{attribute 'linkalways'} 
{attribute 'no_explicit_call' := 'This FB is a CLASS and must be accessed using methods or properties'}
{attribute 'enable_dynamic_creation'}
FUNCTION_BLOCK _ETcVnCircularityCalculationMethod EXTENDS EnumDatatypeBase
VAR
	localData : ETcVnCircularityCalculationMethod;
	activeData : REFERENCE TO ETcVnCircularityCalculationMethod;
	enumBaseDatatype : _DINT(localData);
END_VAR

METHOD PRIVATE AddLocalEnumeration
VAR_INPUT
	Enumeration : T_MAXSTRING;
	Value : ETcVnCircularityCalculationMethod;
END_VAR
AddEnumeration(Enumeration, Value);
END_METHOD

PROPERTY PUBLIC Address : PVOID
GET
Address := ADR(activeData);
END_GET
END_PROPERTY

METHOD PUBLIC ClearReference
VAR_INPUT
END_VAR
activeData REF= localData;
SetBaseDatatypeReference();
END_METHOD

METHOD PUBLIC Clone : I_Datatype
VAR
    pClone : POINTER TO _ETcVnCircularityCalculationMethod;
END_VAR
pClone := __NEW(_ETcVnCircularityCalculationMethod(InitialValue := Value));
Clone := pClone^;
END_METHOD

METHOD FB_init : BOOL
VAR_INPUT
	bInitRetains : BOOL; // if TRUE, the retain variables are initialized (warm start / cold start)
	bInCopyCode : BOOL;  // if TRUE, the instance afterwards gets moved into the copy code (online change)
	InitialValue : ETcVnCircularityCalculationMethod;
END_VAR
localData := InitialValue;
AddBaseDatatype(enumBaseDatatype);
ClearReference();

AddLocalEnumeration('TCVN_CCM_DEFAULT', ETcVnCircularityCalculationMethod.TCVN_CCM_DEFAULT);
AddLocalEnumeration('TCVN_CCM_CONVEXHULL_PERIMETER', ETcVnCircularityCalculationMethod.TCVN_CCM_CONVEXHULL_PERIMETER);
AddLocalEnumeration('TCVN_CCM_MAX_RADIUS', ETcVnCircularityCalculationMethod.TCVN_CCM_MAX_RADIUS);
AddLocalEnumeration('TCVN_CCM_ENCLOSINGCIRCLE_RADIUS', ETcVnCircularityCalculationMethod.TCVN_CCM_ENCLOSINGCIRCLE_RADIUS);
END_METHOD

PROPERTY PUBLIC Identifier : T_MAXSTRING
GET
Identifier := 'ETcVnCircularityCalculationMethod';
END_GET
END_PROPERTY

METHOD IsEnumeratorValueEqual : BOOL
VAR_INPUT
	Enumerator : I_KeyValueForwardEnumerator;
END_VAR
VAR
	storedValue : ETcVnCircularityCalculationMethod;
END_VAR
IF NOT Enumerator.TryGet(storedValue) THEN
	RETURN;
END_IF

IsEnumeratorValueEqual := storedValue = activeData;
END_METHOD

METHOD PUBLIC MakeReferenceTo
VAR_INPUT
	ReferenceTarget : REFERENCE TO ETcVnCircularityCalculationMethod;
END_VAR
activeData REF= ReferenceTarget;
SetBaseDatatypeReference();
END_METHOD

METHOD PROTECTED SetBaseDatatypeReference
VAR_INPUT
END_VAR
enumBaseDatatype.MakeReferenceTo(activeData);
END_METHOD

PROPERTY PUBLIC Size : UDINT
GET
Size := SIZEOF(activeData);
END_GET
END_PROPERTY

METHOD TryMakeReferenceTo : BOOL
VAR_INPUT
	Target : I_Datatype;
END_VAR
VAR
	pTargetData : POINTER TO ETcVnCircularityCalculationMethod;
END_VAR
IF NOT IsEquivalentTo(Target) THEN
	RETURN;
END_IF

pTargetData := Target.Address;
activeData REF= pTargetData^;
SetBaseDatatypeReference();
TryMakeReferenceTo := TRUE;
END_METHOD

PROPERTY PUBLIC Value : ETcVnCircularityCalculationMethod
GET
Value := activeData;
END_GET
SET
activeData := Value;
END_SET
END_PROPERTY

END_FUNCTION_BLOCK

(* stored: Version 1.1.0.1, ProductVersion 3.1.4024.15
   POU _ETcVnCircularityCalculationMethod: Id {873fc11c-d987-0f0c-25a2-9fbc7d322e4d}, SpecialFunc None
   Folder Core: Id {71831f8a-99a3-07c7-1baa-0cc4116a5fcc}
   Folder Protected: Id {0eb4e4bd-b01a-038f-32ba-080c229bf085}
   Folder Customize: Id {11c61f3c-158c-0abb-1080-a1dbeaeec686}
   Folder Constructor: Id {27e27c75-4b10-0985-00fc-add2694d61dd}
   Folder Private: Id {8841fb00-a904-0212-113f-0275a6fea801}
   Folder Protected: Id {fca2cdfd-0dcb-0c9d-3c48-bda33f8d1651}
   Method AddLocalEnumeration: Id {7d1cb6c2-fa7a-01e7-0273-5ec36e377d56}
   Property Address: Id {d3f1de98-508a-036a-040b-9cbe7961f14f}
   Get Get: Id {9ba673cb-d159-0eda-03e9-af5521484749}
   Method ClearReference: Id {a4524275-b9b0-0035-21d1-d17b03de18bf}
   Method Clone: Id {b402053f-0d2a-0838-0a4c-1e4c9ce4f46d}
   Method FB_init: Id {91ca9d31-c2e5-014f-12b3-549374ba36fb}
   Property Identifier: Id {fa5295f2-870e-0bec-37d0-0a5cc8a2b477}
   Get Get: Id {a6e2bac1-2679-0b45-3248-8b96347860da}
   Method IsEnumeratorValueEqual: Id {3680cdf6-2d85-07fe-1e19-6ea98c07b9c6}
   Method MakeReferenceTo: Id {6255410b-eba7-03a5-2e1d-17b34dce431e}
   Method SetBaseDatatypeReference: Id {933bdcf6-d6f1-0981-0564-0787c39d5a13}
   Property Size: Id {2f69cd50-2bfb-00aa-3c76-14579f6b7123}
   Get Get: Id {d8722285-dcf2-0dfa-1c49-18ca9dcdb034}
   Method TryMakeReferenceTo: Id {905b801b-68c0-06c3-0075-04ab6be5c8ac}
   Property Value: Id {edcd1e63-84eb-0a7e-2924-1b0edfcd6df8}
   Get Get: Id {0d966f35-b8ae-0848-0b25-7f2dd45268a7}
   Set Set: Id {c901002d-4324-0b56-21db-041e0ac44e94} *)
